TYPE XML_CONTROL :
STRUCT
	COMMAND : WORD;
	WATCHDOG : TIME;
	START_POS : UINT;
	STOP_POS : UINT;
	COUNT : UINT;
	TYP : INT;
	LEVEL : UINT;
	PATH : STRING(STRING_LENGTH);
	ELEMENT : STRING(STRING_LENGTH);
	ATTRIBUTE : STRING(STRING_LENGTH);
	VALUE : STRING(STRING_LENGTH);
	BLOCK1_START : UINT;
	BLOCK1_STOP : UINT;
	BLOCK2_START : UINT;
	BLOCK2_STOP : UINT;
END_STRUCT
END_TYPE

(* stored: Version 1.1.0.1, ProductVersion 3.1.4022.7
   DUT XML_CONTROL: Id {01ff86ac-2a56-4bba-a82f-05f709ddeaeb} *)
